PROGRAM PRG_3_PMPS_POST
VAR
    fbArbiterIO: FB_SubSysToArbiter_IO;
    bMR1L1_Veto_OUT: BOOL;
    fbVetoArbiter_L1: FB_VetoArbiter;
	//Fast Fault to Aggregate all Group 1 faults
	g_FastFault		:	FB_FastFault();
	g_FastFaultOutput2: INT;
	q_xFastFaultOut: INT;
END_VAR

bMR1L1_Veto_OUT := PMPS_GVL.stCurrentBeamParameters.aVetoDevices[PMPS.L_Stopper.MR1L1_OUT] AND NOT PMPS_GVL.stCurrentBeamParameters.aVetoDevices[PMPS.L_Stopper.MR1L1_IN];

GVL.fbFastFaultOutput1.Execute();
GVL.fbFastFaultOutput1a.Execute();
GVL.fbFastFaultOutput1b.Execute();
GVL.fbFastFaultOutput1c.Execute();
GVL.fbFastFaultOutput1d.Execute();
GVL.fbFastFaultOutput2.Execute(i_xVeto:=bMR1L1_Veto_OUT);

// Aggregate FastFaultOutputs into a single FastFault
g_FastFault(
    io_fbFFHWO := GVL.fbFastFaultOutput1,
    i_xOK := (  GVL.fbFastFaultOutput1a.q_xFastFaultOut
                AND GVL.fbFastFaultOutput1b.q_xFastFaultOut
				AND GVL.fbFastFaultOutput1c.q_xFastFaultOut
				AND GVL.fbFastFaultOutput1d.q_xFastFaultOut
             ),
    i_xAutoReset:=TRUE,
	i_DevName :='Aggregate LFE CC FastFaultOutputs'
);




fbVetoArbiter_L1(bVeto:=bMR1L1_Veto_OUT,
                HigherAuthority := GVL.fbArbiter,
                LowerAuthority := GVL.fbArbiter2,
                FFO := GVL.fbFastFaultOutput1);

fbArbiterIO(
    Arbiter:=GVL.fbArbiter,
    fbFFHWO:=GVL.fbFastFaultOutput1);

END_PROGRAM

(* stored: Version 1.1.0.1
   POU PRG_3_PMPS_POST: Id {ae2b5b23-f406-4591-b6ea-00080d408961}, SpecialFunc None *)
